FUNCTION_BLOCK L3_ReceivePart (* Basic Function Block Type *)
  (* Standard: 61499-2 *)
  (* Version 0.0, 2014-10-02, EQUEROL, UJI *)
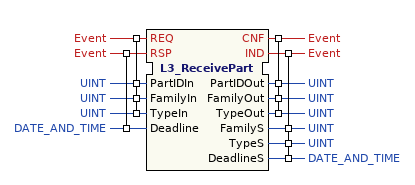
  EVENT_INPUT
    REQ WITH PartIDIn, FamilyIn, TypeIn; (* Normal Execution Request *)
    RSP WITH Deadline; (* Response, Part correctly added *)
  END_EVENT
  EVENT_OUTPUT
    CNF WITH PartIDOut, FamilyOut, TypeOut; (* Execution Confirmation *)
    IND WITH DeadlineS, TypeS, FamilyS; (* Indicate that part was correctly added *)
  END_EVENT
  VAR_INPUT
    PartIDIn : UINT; (* Part's identifier *)
    FamilyIn : UINT; (* Part's family *)
    TypeIn : UINT; (* Part's type *)
    Deadline : DATE_AND_TIME;
  END_VAR
  VAR_OUTPUT
    PartIDOut : UINT; (* Part's identifier *)
    FamilyOut : UINT; (* Part's family *)
    TypeOut : UINT; (* Part's type *)
    FamilyS : UINT; (* Part's family *)
    TypeS : UINT; (* Part's type *)
    DeadlineS : DATE_AND_TIME; (* Updated deadline for this pair family-type *)
  END_VAR
  VAR
    CurrentID : UINT; (* ID of the part being updated *)
    CurrentFamily : UINT; (* Family of the part being updated *)
    CurrentType : UINT; (* Type of the part being updated *)
    LostIND : BOOL; (* Internal Variable *)
    CompletedIDS : ARRAY [0..24] OF UINT := [0,0,0,0,0,0,0,0,0,0,0,0,0,0,0,0,0,0,0,0,0,0,0,0,0]; (* Circular buffer *)
    CompletedFamilies : ARRAY [0..24] OF UINT; (* Circular buffer *)
    CompletedTypes : ARRAY [0..24] OF UINT; (* Circular buffer *)
    CompletedDeadlines : ARRAY [0..24] OF DATE_AND_TIME; (* Circular buffer *)
    Index : UINT := 0; (* Completed actions vector Index. Points to the oldest entry in the vector *)
    i : UINT; (* boucle variable *)
  END_VAR
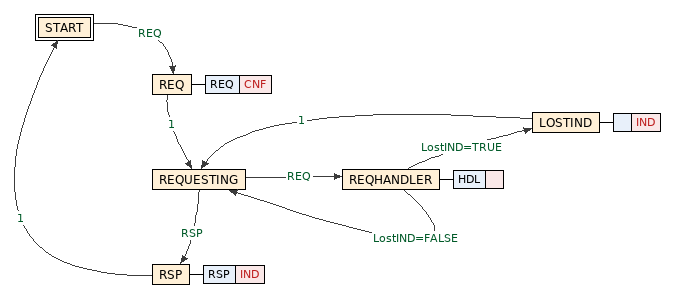
  EC_STATES
    START; (* Initial State *)
    REQ : REQ -> CNF; (* Normal execution *)
    REQUESTING;
    REQHANDLER : HDL;
    LOSTIND : -> IND;
    RSP : RSP -> IND;
  END_STATES
  EC_TRANSITIONS
    START TO REQ := REQ;
    REQUESTING TO RSP := RSP;
    REQ TO REQUESTING := 1;
    RSP TO START := 1;
    REQUESTING TO REQHANDLER := REQ;
    LOSTIND TO REQUESTING := 1;
    REQHANDLER TO LOSTIND := LostIND=TRUE;
    REQHANDLER TO REQUESTING := LostIND=FALSE;
  END_TRANSITIONS
  ALGORITHM REQ IN ST: (* Normally executed algorithm *)
(*Update current action data*)
CurrentID := PartIDIn;
CurrentFamily := FamilyIn;
CurrentType := TypeIn;
(*Map input to output*)
PartIDOut := PartIDIn;
FamilyOut := FamilyIn;
TypeOut := TypeIn;
  END_ALGORITHM
  ALGORITHM HDL IN ST: (* Algorithm to handle lost IND and Timeouts while receiving IND *)
(*New request arrived while processing one*)
(*Verify if the request is a previously completed action*)
i := 0;
LostIND := FALSE;
WHILE (i < 25 )DO
	IF ( PartIDIn =CompletedIDS[i] ) THEN
		(*Received request has already been processed*)
		(*Send IND*)
		LostIND := TRUE;
		(*Update output values*)
		FamilyS := CompletedFamilies[i];
		TypeS := CompletedTypes[i];
		DeadlineS := CompletedDeadlines[i];
		(*exit loop*)
		i := 26;
	ELSE
		i := i + 1;
	END_IF;
END_WHILE;
  END_ALGORITHM
  ALGORITHM RSP IN ST: (* algorithm to register completed actions *)
(*Completed Action*)
CompletedIDS[Index] := CurrentID;
CompletedFamilies[Index] := CurrentFamily;
CompletedTypes[Index] := CurrentType;
CompletedDeadlines[Index] := Deadline;

(*Increase Index*)
Index :=mod(Index+1, 25);

(*Map input to output*)
FamilyS := CurrentFamily;
TypeS := CurrentType;
DeadlineS := Deadline;
  END_ALGORITHM
END_FUNCTION_BLOCK
